Staubli VAL3: remErrPPTimeout.pgx

program remErrPpTimeout(num& nTime[] (dimensions=1), string& sReturn[] (dimensions=1))
begin
  // Error raised when waiting for PPS ready times out
  //
  logMsg("call remErrTimeout")
  sReturn="ERROR 901"
  sReturn=sReturn+": Timeout of PPS ready after "
  sReturn=sReturn+toString("",nTime)+" seconds."
  putln(sReturn)
  logMsg(sReturn)
end
